FUNCTION_BLOCK TestStruct2TestStruct (* Basic Function Block Type *)
  (* Standard: 61499-2 *)
  (* Version 0.9, 2012-01-10, IH, 4DIAC *)
  (* Compiler header: package fb.rt.test; import fb.rt.test.TestStruct; *)
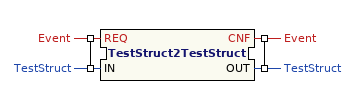
  EVENT_INPUT
    REQ WITH IN; (* Normal Execution Request *)
  END_EVENT
  EVENT_OUTPUT
    CNF WITH OUT; (* Execution Confirmation *)
  END_EVENT
  VAR_INPUT
    IN : TestStruct; (* Input *)
  END_VAR
  VAR_OUTPUT
    OUT : TestStruct; (* Output *)
  END_VAR
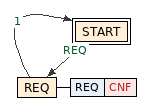
  EC_STATES
    START; (* Initial State *)
    REQ : REQ -> CNF; (* Normal execution *)
  END_STATES
  EC_TRANSITIONS
    START TO REQ := REQ;
    REQ TO START := 1;
  END_TRANSITIONS
  ALGORITHM REQ IN Java: (* Normally executed algorithm *)
OUT.FOO.value=IN.FOO.value;
OUT.BAR.value=IN.BAR.value;
  END_ALGORITHM
END_FUNCTION_BLOCK
